FUNCTION_BLOCK basicIOComGate (* Gate de comunicacao de remota Modbus: zera as words e sinaliza falha quando a remota esta offline *)
  (* Standard: 61499-2 *)
  (* Version 1.0, 10/2/2026, Hidryco, Hidryco, Criado para IO_DI32 e IO_DQ32 *)
  PACKAGE Hidryco.HidrycoLib;
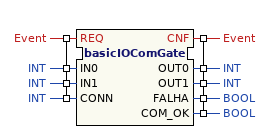
  EVENT_INPUT
    REQ WITH IN0, IN1, CONN; (* Nova leitura das words ou do status de comunicacao *)
  END_EVENT
  EVENT_OUTPUT
    CNF WITH OUT0, OUT1, FALHA, COM_OK; (* Saidas atualizadas *)
  END_EVENT
  VAR_INPUT
    IN0 : INT; (* Word 0 lida da remota *)
    IN1 : INT; (* Word 1 lida da remota *)
    CONN : INT; (* connStatusInt do acoplador: 1 online, 0 offline *)
  END_VAR
  VAR_OUTPUT
    OUT0 : INT; (* Word 0 liberada (0 se offline) *)
    OUT1 : INT; (* Word 1 liberada (0 se offline) *)
    FALHA : BOOL; (* TRUE = remota offline *)
    COM_OK : BOOL; (* TRUE = remota online *)
  END_VAR
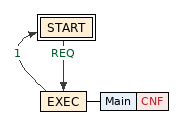
  EC_STATES
    START; (* Initial State *)
    EXEC : Main -> CNF;
  END_STATES
  EC_TRANSITIONS
    START TO EXEC := REQ;
    EXEC TO START := 1;
  END_TRANSITIONS
  ALGORITHM Main IN ST: (* Gate de comunicacao *)
(* Libera as words da remota somente com a comunicacao OK.
   CONN = connStatusInt do acoplador Modbus (1 = online, 0 = offline).
   Remota offline: words = 0 (todos os bits FALSE) e FALHA = TRUE. *)
IF CONN = 1 THEN
    OUT0 := IN0;
    OUT1 := IN1;
    FALHA := FALSE;
ELSE
    OUT0 := 0;
    OUT1 := 0;
    FALHA := TRUE;
END_IF;
COM_OK := NOT FALHA;
  END_ALGORITHM
END_FUNCTION_BLOCK
